{attribute 'Tc2GvlVarNames'}
VAR_CONFIG
END_VAR

(* stored: Version 1.1.0.1, ProductVersion 3.1.4024.3
   GVL Variablen_Konfiguration: Id {7935c8aa-422c-4d72-bb9f-3f1aced7cbe0} *)
